RoboDK station: HAMK_Vacuum_gripper_MG400.rdk

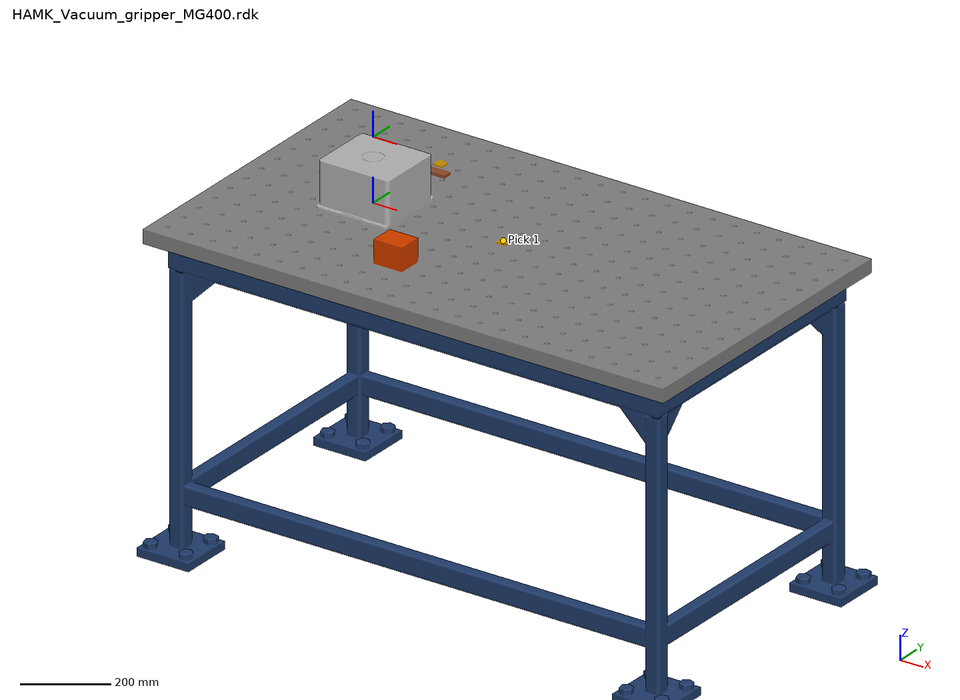
[picture v0: the station drawn from its stored meshes, robots at their saved joint values, targets as dots, program paths as lines]
Station HAMK_Vacuum_gripper_MG400 (saved by RoboDK 5.8.0). Poses are relative to the parent item; angles as X-Y-Z fixed-axis rotations.
Station parameters (name, value as stored): IO_1, 1, IO_5, 1
  - frame Dobot MG400 Base at (0, 0, 0) mm
    - robot Dobot MG400: 4 axes, payload 0.5 kg, reach 393.5 mm, repeatability 0.2 mm, weight 4 kg
        joint limits [-160, -25, -25, -360] to [160, 85, 105, 360]; home [0, 0, 0, 0]; saved at [0, 72.531, 65.14, 180]
      - tool Suction Cup, TCP at (0, 0, -76) mm, size 42.6 x 40 x 76.8 mm
    - frame World at (0, 0, 0) mm
      - object Table 1400x800x800mm at (0, 0, 0) mm, size 1420 x 820 x 800 mm, geometry from Table-1400x800x800mm.sld
        - object HAMK logo at (360, 380, -115) mm, rotated rx 90 ry 0 rz 180 deg, size 301.4 x 100.9 x 9.4 mm, geometry from Fantastic Duup(2).stl
        - object white background at (360, 385.5, -110) mm, rotated rx 90 ry 0 rz 0 deg, size 480 x 184.8 x 2.4 mm, geometry from Fantastic Duup(3).stl
      - object Kapla wood block 0 at (0, 200, 0) mm, size 117 x 23.4 x 7.8 mm, geometry from Kapla wood block.stl
      - object Box at (176, -250, 0) mm, size 76 x 62 x 60 mm, geometry from cube.sld
      - object Mosaic title 0 at (0, 230, 0) mm, size 24 x 24 x 4 mm, geometry from cube.sld
      - object Mosaic title 1 at (338.5, -12, 0) mm, size 24 x 24 x 4 mm, geometry from cube.sld
  - frame RefSuctionCup at (0, 0, 161.75) mm
    - target Pick 1 (Cartesian target) at (350, 0, -157) mm; joints [0, 72.531, 65.14, 180] of Dobot MG400
